Fanuc KAREL source: kt00335.KL

PROGRAM KT00335
%STACKSIZE=65535
%PRIORITY=65535
%NOLOCKGROUP
VAR
R1 : REAL
OUT : BOOLEAN
-- UNRESOLVED DECLARATIONS (source type spelling not recovered)
-- Y2 : ARRAY[2] OF TYPE_0x0018 (type_u16=0x2018)
BEGIN
R1=2.0
Y2[1]=3
-- UNRESOLVED_PC line 10 opcodes [21 22 9D 33 B1 64 6F 23] marker_code=35
END KT00335
